# EPICS substitutions: iocBoot/iocStdTest/selector.substitutions
file "$(STD)/stdApp/Db/selector.db"
{
{P=stdTest:,    R=obj,
NAME1="5x",  PV1="$(P)m1.VAL", VAL1=3,
NAME2="10x", PV2="$(P)m1.VAL", VAL2=6,
NAME3="20x", PV3="$(P)m1.VAL", VAL3=9
}
}
